{attribute addProperty BoxType "CU1123-0000-0016"}
{attribute addProperty Id "A_0002_CU1123_0010_0016A_0002_CU1123_0010_0016_1433E11E992124"}
{attribute addProperty CRC "1850495919"}
{attribute addProperty SizeInBites "992"}
{attribute addProperty SizeInBytes "124"}
TYPE A_0001_CU1123_0000_0016_6E4C53AF EXTENDS CU1123_179A0949 :
STRUCT
	{attribute addProperty Name "A_0002_CU1123_0010_0016"}
	A_0002_CU1123_0010_0016 : A_0002_CU1123_0010_0016_1433E11E;
END_STRUCT
END_TYPE

(* stored: Version 1.2.0.0, ProductVersion 3.1.4024.9
   DUT A_0001_CU1123_0000_0016_6E4C53AF: Id {39955574-9498-46f1-93ff-500f1db5a3a8} *)
